FUNCTION_BLOCK SUBL_TEST (* Test SUBL_x in a Composite Function Block *)
  (* Standard: 61499-2 *)
  (* Version 0.0, 2002-12-17, JHC, RA *)
  (* Compiler header: package fb.rt.test; import fb.rt.net.*; *)
  (* Compiler Java IBM Jikes 1.06 *)
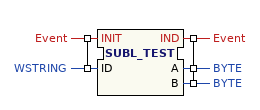
  EVENT_INPUT
    INIT WITH ID;
  END_EVENT
  EVENT_OUTPUT
    IND WITH A, B;
  END_EVENT
  VAR_INPUT
    ID : WSTRING;
  END_VAR
  VAR_OUTPUT
    A : BYTE;
    B : BYTE;
  END_VAR
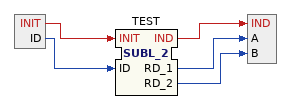
  FBS
    TEST : SUBL_2;
  END_FBS
  EVENT_CONNECTIONS
    INIT TO TEST.INIT;
    TEST.IND TO IND;
  END_CONNECTIONS
  DATA_CONNECTIONS
    ID TO TEST.ID;
    TEST.RD_1 TO A;
    TEST.RD_2 TO B;
  END_CONNECTIONS
END_FUNCTION_BLOCK
